FUNCTION_BLOCK Service_AOControl (* Basic Function Block Type *)
  (* Standard: 61499-2 *)
  (* Version 0.0, 2014-5-4, wildai, nxtControl GmbH, Template *)
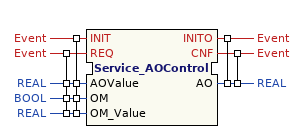
  EVENT_INPUT
    INIT WITH AOValue, OM, OM_Value; (* Initialization Request *)
    REQ WITH AOValue, OM, OM_Value; (* Normal Execution Request *)
  END_EVENT
  EVENT_OUTPUT
    INITO WITH AO; (* Initialization Confirm *)
    CNF WITH AO; (* Execution Confirmation *)
  END_EVENT
  VAR_INPUT
    AOValue : REAL;
    OM : BOOL;
    OM_Value : REAL;
  END_VAR
  VAR_OUTPUT
    AO : REAL;
  END_VAR
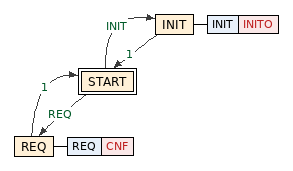
  EC_STATES
    START; (* Initial State *)
    INIT : INIT -> INITO; (* Initialization *)
    REQ : REQ -> CNF; (* Normal execution *)
  END_STATES
  EC_TRANSITIONS
    START TO INIT := INIT;
    INIT TO START := 1;
    START TO REQ := REQ;
    REQ TO START := 1;
  END_TRANSITIONS
  ALGORITHM INIT IN ST: (* Initialization algorithm *)
;
AO := 0.0;
  END_ALGORITHM
  ALGORITHM REQ IN ST: (* Normally executed algorithm *)
;

IF OM THEN
	AO := OM_Value;
ELSE
	AO := AOValue;
END_IF;
  END_ALGORITHM
END_FUNCTION_BLOCK
